// TwinCAT 3 PLC project rplc
// Title: rplc
// Company: TcHaxx
// Author: densogiaichned
// ProjectVersion: 0.3.2.0
// Description: Invoke RPC methods.
// ProgramVersion: 3.1.4024.0
// libraries:
//   Tc2_Standard, * (Beckhoff Automation GmbH)
//   Tc2_System, * (Beckhoff Automation GmbH)
//   Tc3_Module, * (Beckhoff Automation GmbH)
//   TcUnit, * (www.tcunit.org)
// project tree:
//   DUTs/ ST_AdsStatus.TcDUT, ST_AnyType.TcDUT
//   GVLs/ GCL.TcGVL, Param_Args.TcGVL
//   ITFs/ I_ArgsBuffer.TcIO, I_RpcArguments.TcIO, I_RpcDynamicConfigAmsNetId.TcIO, I_RpcDynamicConfigAmsPort.TcIO, I_RpcDynamicConfigSymbolPath.TcIO, I_RpcDynamicConfig.TcIO, I_RpcDynamicConfigBuild.TcIO, I_RpcInvoke.TcIO, I_RpcReleaseHandle.TcIO
//   / PlcTaskUnitTest.TcTTO
//   POUs/ FB_RPC.TcPOU, FB_RPC_Dynamic.TcPOU, F_ToAnyType.TcPOU
//   POUs/internal/ FB_ArgumentsBuffer.TcPOU, FB_RpcConfig.TcPOU, FB_RpcBase.TcPOU, F_RpcSymbol.TcPOU (not stored)
//   TESTs/ FB_F_RpcSymbol_Tests.TcPOU, FB_F_ToAnyType_Tests.TcPOU, FB_RPC_Tests.TcPOU, FB_RPC_Dynamic_Tests.TcPOU, PRG_UnitTests.TcPOU
//   TESTs/Helper/ E_Mode.TcDUT, F_IncrementStep.TcPOU
// real-time tasks:
//   TASK PlcTask: cycle T#10ms, priority 20, ADS port 350
//   TASK PlcTaskUnitTest: cycle T#10ms, priority 1, ADS port 351
//   TASK PlcTaskRpcServer: cycle T#10ms, priority 21, ADS port 352
//   TASK PlcTaskRpcClient: cycle T#10ms, priority 22, ADS port 353

CONFIGURATION rplc
    RESOURCE PLC ON TwinCAT3
        TASK PlcTaskUnitTest(INTERVAL := T#10ms, PRIORITY := 1);
        PROGRAM PRG_UnitTests WITH PlcTaskUnitTest : PRG_UnitTests;
    END_RESOURCE
END_CONFIGURATION

// ---- DUTs/ST_AdsStatus.TcDUT
{attribute 'pack_mode' = '1'}
TYPE ST_AdsStatus :
STRUCT
	bBusy	: BOOL;
	bError	: BOOL;
	nError 	: UDINT;
END_STRUCT
END_TYPE

// ---- DUTs/ST_AnyType.TcDUT
{attribute 'pack_mode' = '1'}
TYPE ST_AnyType :
STRUCT
	pValue : PVOID;
	nSize  : DINT;
	TypeClass : __SYSTEM.TYPE_CLASS;
END_STRUCT
END_TYPE

// ---- TESTs/Helper/E_Mode.TcDUT
{attribute 'qualified_only'}
{attribute 'strict'}
TYPE E_Mode :
(
	BUSY := 0,
	INC := 1,
	END := 99
);
END_TYPE

// ---- GVLs/GCL.TcGVL
{attribute 'qualified_only'}
{attribute 'no-analysis'}
{attribute 'global_init_slot' := '49991'}
VAR_GLOBAL CONSTANT
	cLocalAmsNetId		: STRING := '127.0.0.1.1.1';
	cAdsTimeOut			: TIME := Tc2_System.DEFAULT_ADS_TIMEOUT;
	cRpcSymbolSeparator : STRING := '#';
END_VAR

// ---- GVLs/Param_Args.TcGVL
{attribute 'qualified_only'}
{attribute 'no-analysis'}
VAR_GLOBAL CONSTANT
	cMaxArgsBuffer		: UDINT(64..1048576) 	:= 65536;	// max sizeof aArgs buffer array in bytes.
	cMaxArgs			: USINT(1..128) 		:= 32;		// max length method arguments
END_VAR

// ---- ITFs/I_ArgsBuffer.TcIO
INTERFACE I_ArgsBuffer

PROPERTY nArgsLength : UDINT
GET
END_GET
END_PROPERTY

PROPERTY nRetValLength : UDINT
GET
END_GET
END_PROPERTY

PROPERTY pArgsBuffer : POINTER TO BYTE
GET
END_GET
END_PROPERTY

PROPERTY pRetValBuffer : POINTER TO BYTE
GET
END_GET
END_PROPERTY

END_INTERFACE

// ---- ITFs/I_RpcArguments.TcIO
INTERFACE I_RpcArguments

METHOD NoReturnValue : I_RpcInvoke
VAR_INPUT
END_VAR
END_METHOD

METHOD ReturnValue : I_RpcInvoke
VAR_INPUT
	anyRetVal	: ANY;
END_VAR
END_METHOD

METHOD VarInOut : I_RpcArguments
VAR_INPUT
	anyArg	: ANY;
END_VAR
END_METHOD

METHOD VarInput : I_RpcArguments
VAR_INPUT
	anyArg	: ANY;
END_VAR
END_METHOD

METHOD VarOutput : I_RpcArguments
VAR_INPUT
	anyArg	: ANY;
END_VAR
END_METHOD

END_INTERFACE

// ---- ITFs/I_RpcDynamicConfigAmsNetId.TcIO
INTERFACE I_RpcDynamicConfigAmsNetId

METHOD WithAmsNetId : I_RpcDynamicConfigAmsPort
VAR_INPUT
	sAmsNetId	: T_AmsNetID;
END_VAR
END_METHOD

END_INTERFACE

// ---- ITFs/I_RpcDynamicConfigAmsPort.TcIO
INTERFACE I_RpcDynamicConfigAmsPort

METHOD WithAmsPort : I_RpcDynamicConfigSymbolPath
VAR_INPUT
	nAmsPort	: T_AmsPort;
END_VAR
END_METHOD

END_INTERFACE

// ---- ITFs/I_RpcDynamicConfigSymbolPath.TcIO
INTERFACE I_RpcDynamicConfigSymbolPath

METHOD WithSymbolPath : I_RpcDynamicConfigBuild
VAR_INPUT
	sInstancePath	: STRING;
	sSymbol			: STRING;
END_VAR
END_METHOD

END_INTERFACE

// ---- ITFs/I_RpcDynamicConfig.TcIO
INTERFACE I_RpcDynamicConfig

METHOD Configure : I_RpcDynamicConfigAmsNetId
VAR_INPUT
END_VAR
END_METHOD

END_INTERFACE

// ---- ITFs/I_RpcDynamicConfigBuild.TcIO
INTERFACE I_RpcDynamicConfigBuild

METHOD Build : HRESULT
VAR_INPUT
END_VAR
END_METHOD

END_INTERFACE

// ---- ITFs/I_RpcInvoke.TcIO
INTERFACE I_RpcInvoke

METHOD Invoke : ST_AdsStatus
VAR_INPUT
END_VAR
END_METHOD

END_INTERFACE

// ---- ITFs/I_RpcReleaseHandle.TcIO
INTERFACE I_RpcReleaseHandle

METHOD ReleaseHandle : ST_AdsStatus
VAR_INPUT
END_VAR
END_METHOD

END_INTERFACE

// ---- TESTs/PRG_UnitTests.TcPOU
{attribute 'analysis' := '-33'}
PROGRAM INTERNAL PRG_UnitTests

VAR
{IF defined (UNIT_TEST)}	
	fbF_RpcSymbolTests			: FB_F_RpcSymbol_Tests;
	fbRpcTests					: FB_RPC_Tests;
	fbRpcDynamicTests			: FB_RPC_Dynamic_Tests;
	fbF_ToAnyTypeTests			: FB_F_ToAnyType_Tests;
{END_IF}
END_VAR

{IF defined (UNIT_TEST)}
TcUnit.RUN();
{END_IF}

END_PROGRAM

// ---- TESTs/FB_F_RpcSymbol_Tests.TcPOU
{attribute 'reflection'}
FUNCTION_BLOCK INTERNAL FINAL FB_F_RpcSymbol_Tests EXTENDS TcUnit.FB_TestSuite
VAR_INPUT
END_VAR
VAR_OUTPUT
END_VAR
VAR
	{attribute 'instance-path'} 
    {attribute 'noinit'} 
	sTestName			: T_MaxString;
	sActual				: T_MaxString;
	sMaxString			: T_MaxString := 'iwgNivAMcHfLkBpkvqNXNWYnMrQNVzUhZFVRYSjRcjnJtRacqFJhzGPkUNrHkvVpMnnxcBtbBwcrvBgfHgaLBQffiYTVjMkCQgidjvwmnvQEQCzVzZUguBPbnEQCfVDbiCMwiEdfqETncfBwbYbhTrSuRhWzNxVpQzBiWeHAGjdWTLmVfyFKEWMhmMgWqFvtAhBarrEkqQCMJvWxGcDZUfMZwdEebgjfuXXMJwGbgzpjyqzigwxkZiHXPvZCmcn';
END_VAR


TEST(sTestName);

TEST('Should build RPC symbol successfully');

sActual := F_RpcSymbol('', '');
AssertEquals_STRING(Expected:= GCL.cRpcSymbolSeparator,
					Actual:= sActual,
					Message:= 'Expected # only');

sActual := F_RpcSymbol('abc', '');
AssertEquals_STRING(Expected:= 'abc#',
					Actual:= sActual,
					Message:= 'Expected abc# only');

sActual := F_RpcSymbol('', 'abc');
AssertEquals_STRING(Expected:= '#abc',
					Actual:= sActual,
					Message:= 'Expected #abc only');

sActual := F_RpcSymbol('InstancePath', 'SymbolName');
AssertEquals_STRING(Expected:= 'InstancePath#SymbolName',
					Actual:= sActual,
					Message:= 'Expected InstancePath#SymbolName');
TEST_FINISHED();

TEST('Should return sInstancePath if > T_MaxString');

sActual := F_RpcSymbol(sMaxString, 'abc');
AssertEquals_STRING(Expected:= sMaxString,
					Actual:= sActual,
					Message:= 'Expected sInstancePath');
TEST_FINISHED();

TEST('Should truncate if > T_MaxString');


sActual := F_RpcSymbol('abc', sMaxString);
AssertEquals_STRING(Expected:= CONCAT('abc#', LEFT(sMaxString, 251)),
					Actual:= sActual,
					Message:= 'Expected abc#iwgNivAMcHfLk...ZiHXPvZ');
TEST_FINISHED();

TEST_FINISHED_NAMED(sTestName);

END_FUNCTION_BLOCK

// ---- TESTs/FB_RPC_Tests.TcPOU
{attribute 'reflection'}
FUNCTION_BLOCK INTERNAL FINAL FB_RPC_Tests EXTENDS TcUnit.FB_TestSuite
VAR
	{attribute 'instance-path'} 
    {attribute 'noinit'} 
	sTestName			: T_MaxString;
	sActiveStep			: T_MaxString;
	nSequence			: INT;
	nSeqOld				: INT;
	nRpcMethodInvoked 	: UDINT;
	aSUTs				: ARRAY[0..255] OF I_RpcReleaseHandle;
END_VAR
VAR_TEMP
	eMode	: E_Mode;
END_VAR

CASE nSequence OF
	0:
		TEST(sTestName);
		F_IncrementStep(nStepToInc:= nSequence, sActiveStep:= sActiveStep, eMode:= E_Mode.INC);
	1:
		sActiveStep := 'ShouldInvokeMethod_NoArguments_NoReturnValue_Successfully';
		TEST(sActiveStep);
		eMode := ShouldInvokeMethod_NoArguments_NoReturnValue_Successfully();
		F_IncrementStep(nStepToInc:= nSequence, sActiveStep, eMode);
	2:
		sActiveStep := 'ShouldInvokeMethod_NoArguments_ReturnValueBoolean_Successfully';
		TEST(sActiveStep);
		eMode := ShouldInvokeMethod_NoArguments_ReturnValueBoolean_Successfully();
		F_IncrementStep(nStepToInc:= nSequence, sActiveStep, eMode);
	3:	
		sActiveStep := 'ShouldInvokeMethod_OneArgument_NoReturnValue_Successfully';
		TEST(sActiveStep);
		eMode := ShouldInvokeMethod_OneArgument_NoReturnValue_Successfully();
		F_IncrementStep(nStepToInc:= nSequence, sActiveStep, eMode);	
	4:	
		sActiveStep := 'ShouldInvokeMethod_OneArgument_NoReturnValue_Successfully';
		TEST(sActiveStep);
		eMode := ShouldInvokeMethod_OneArgument_NoReturnValue_Successfully();
		F_IncrementStep(nStepToInc:= nSequence, sActiveStep, eMode);	
	5:	
		sActiveStep := 'ShouldInvokeMethod_TwoArguments_ReturnValue_Successfully';
		TEST(sActiveStep);
		eMode := ShouldInvokeMethod_TwoArguments_ReturnValue_Successfully();
		F_IncrementStep(nStepToInc:= nSequence, sActiveStep, eMode);
	6:	
		sActiveStep := 'ShouldInvokeMethod_ThreeArguments_ReturnValue_Successfully';
		TEST(sActiveStep);
		eMode := ShouldInvokeMethod_ThreeArguments_ReturnValue_Successfully();
		F_IncrementStep(nStepToInc:= nSequence, sActiveStep, eMode);		
	7:	
		sActiveStep := 'ShouldInvokeMethod_VarInOutConstant_ReturnValue_Successfully';
		TEST(sActiveStep);
		eMode := ShouldInvokeMethod_VarInOutConstant_ReturnValue_Successfully();
		F_IncrementStep(nStepToInc:= nSequence, sActiveStep, eMode);	
	8:	
		sActiveStep := 'ShouldInvokeMethod_VarOutput_ReturnValue_Successfully';
		TEST(sActiveStep);
		eMode := ShouldInvokeMethod_VarOutput_ReturnValue_Successfully();
		F_IncrementStep(nStepToInc:= nSequence, sActiveStep, eMode);	
	9:	
		sActiveStep := 'ShouldInvokeMethod_TwoVarOutput_ReturnValue_Successfully';
		TEST(sActiveStep);
		eMode := ShouldInvokeMethod_TwoVarOutput_ReturnValue_Successfully();
		F_IncrementStep(nStepToInc:= nSequence, sActiveStep, eMode);	
	10:	
		sActiveStep := 'ShouldInvokeMethod_VarInput_VarInOut_VarOutput_ReturnValue_Successfully';
		TEST(sActiveStep);
		eMode := ShouldInvokeMethod_VarInput_VarInOut_VarOutput_ReturnValue_Successfully();
		F_IncrementStep(nStepToInc:= nSequence, sActiveStep, eMode);		
	11: 
		sActiveStep := 'ShouldReturnError0x705';
		TEST(sActiveStep);
		eMode := ShouldReturnError0x705();
		F_IncrementStep(nStepToInc:= nSequence, sActiveStep, eMode);	
	12: 
		sActiveStep := 'ShouldReturnError0x710';
		TEST(sActiveStep);
		eMode := ShouldReturnError0x710();
		F_IncrementStep(nStepToInc:= nSequence, sActiveStep, eMode);	
	13: 
		sActiveStep := 'ShouldReleaseAllSymbolHandleSuccessfully';
		TEST(sActiveStep);
		eMode := ShouldReleaseAllSymbolHandleSuccessfully();
		F_IncrementStep(nStepToInc:= nSequence, sActiveStep, eMode);	
	ELSE
		TEST_FINISHED_NAMED(sTestName);
END_CASE

IF nSequence <> nSeqOld THEN
	nRpcMethodInvoked := 0;
	nSeqOld := nSequence;
END_IF;

{attribute 'TcRpcEnable'}
METHOD NoParameter_NoReturnValue

nRpcMethodInvoked := nRpcMethodInvoked + 1;
END_METHOD

{attribute 'TcRpcEnable'}
METHOD NoParameter_ReturnValue : BOOL
VAR_INPUT
END_VAR
nRpcMethodInvoked := nRpcMethodInvoked + 1;
NoParameter_ReturnValue := nRpcMethodInvoked > 0;
END_METHOD

{attribute 'TcRpcEnable'}
METHOD OneParameter_NoReturnValue
VAR_INPUT
	nArg1 	: UDINT;
END_VAR
nRpcMethodInvoked := nArg1;
END_METHOD

METHOD Register
VAR_INPUT
	ipRpcReleaseHandle	: I_RpcReleaseHandle;
END_VAR

VAR
	i :UINT;
END_VAR


FOR i:=0 TO 255 DO	
	IF aSUTs[i] = ipRpcReleaseHandle THEN
		EXIT;
	END_IF
	IF aSUTs[i] <> NULL THEN
		CONTINUE;
	END_IF
	
	aSUTs[i] := ipRpcReleaseHandle;
	EXIT;
END_FOR
END_METHOD

METHOD ShouldInvokeMethod_NoArguments_NoReturnValue_Successfully : E_Mode

VAR_INST
	fbSUT		: FB_RPC(GCL.cLocalAmsNetId, _AppInfo.AdsPort, 'PRG_UnitTests.fbRpcTests', 'NoParameter_NoReturnValue');
END_VAR

VAR
	stRetVal	: ST_AdsStatus;
	eMode		: E_Mode := E_MODE.BUSY;
END_VAR
// Arrange
Register(fbSUT);

// Act
stRetVal := fbSUT.Invoke();

IF NOT stRetVal.bBusy THEN
	eMode := E_Mode.INC;
	
	// Assert
	AssertFalse(Condition:= stRetVal.bError, Message:= 'Expected method NoParameter_NoReturnValue to return no error.');
	AssertEquals_UDINT(Expected:= E_AdsErr.NOERR, Actual:= stRetVal.nError, Message:= 'Expected method NoParameter_NoReturnValue to return no error.');
	AssertEquals_UDINT(Expected:= 1, Actual:= nRpcMethodInvoked, Message:= 'Expected method NoParameter_NoReturnValue to be invoked once.');
END_IF

ShouldInvokeMethod_NoArguments_NoReturnValue_Successfully := eMode;
END_METHOD

METHOD ShouldInvokeMethod_NoArguments_ReturnValueBoolean_Successfully : E_Mode

VAR_INST
	fbSUT		: FB_RPC(GCL.cLocalAmsNetId, _AppInfo.AdsPort, 'PRG_UnitTests.fbRpcTests', 'NoParameter_ReturnValue');
END_VAR

VAR
	stRetVal	: ST_AdsStatus;
	eMode		: E_Mode := E_MODE.BUSY;
	bActual		: BOOL;
END_VAR
// Arrange
Register(fbSUT);

// Act
stRetVal := fbSUT.ReturnValue(bActual).Invoke();

IF NOT stRetVal.bBusy THEN
	eMode := E_Mode.INC;
	// Assert
	AssertFalse(Condition:= stRetVal.bError, Message:= 'Expected method NoParameter_ReturnValue to return no error.');
	AssertEquals_UDINT(Expected:= E_AdsErr.NOERR, Actual:= stRetVal.nError, Message:= 'Expected method NoParameter_ReturnValue to return no error.');
	AssertEquals_UDINT(Expected:= 1, Actual:= nRpcMethodInvoked, Message:= 'Expected method NoParameter_ReturnValue to be invoked once.');
	AssertTrue(Condition:= bActual, Message:= 'Expected method NoParameter_ReturnValue to return TRUE.');
END_IF

ShouldInvokeMethod_NoArguments_ReturnValueBoolean_Successfully := eMode;
END_METHOD

METHOD ShouldInvokeMethod_OneArgument_NoReturnValue_Successfully : E_Mode

VAR_INST
	fbSUT		: FB_RPC(GCL.cLocalAmsNetId, _AppInfo.AdsPort, 'PRG_UnitTests.fbRpcTests', 'OneParameter_NoReturnValue');
END_VAR

VAR
	stRetVal	: ST_AdsStatus;
	eMode		: E_Mode := E_MODE.BUSY;
	nArg		: UDINT;
END_VAR
// Arrange
Register(fbSUT);
nArg := 123;

// Act
stRetVal := fbSUT.VarInput(nArg).NoReturnValue().Invoke();

IF NOT stRetVal.bBusy THEN
	eMode := E_Mode.INC;
	
	// Assert
	AssertFalse(Condition:= stRetVal.bError, Message:= 'Expected method OneParameter_NoReturnValue to return no error.');
	AssertEquals_UDINT(Expected:= E_AdsErr.NOERR, Actual:= stRetVal.nError, Message:= 'Expected method OneParameter_NoReturnValue to return no error.');
	AssertEquals_UDINT(Expected:= nArg, Actual:= nRpcMethodInvoked, Message:= 'Expected method OneParameter_NoReturnValue to be invoked with value 123.');
END_IF

ShouldInvokeMethod_OneArgument_NoReturnValue_Successfully := eMode;
END_METHOD

METHOD ShouldInvokeMethod_ThreeArguments_ReturnValue_Successfully : E_Mode

VAR_INST
	fbSUT		: FB_RPC(GCL.cLocalAmsNetId, _AppInfo.AdsPort, 'PRG_UnitTests.fbRpcTests', 'ThreeParameters_ReturnValue');
END_VAR

VAR
	stRetVal	: ST_AdsStatus;
	eMode		: E_Mode := E_MODE.BUSY;
	nArg1		: UDINT;
	stArg2		: ST_AdsStatus;	// IN_OUT!
	sArg3		: STRING;
	sActualRetVal : STRING;
END_VAR
// Arrange
Register(fbSUT);
nArg1 := 456;
stArg2.bBusy := FALSE;
stArg2.bError := TRUE;
stArg2.nError := 321;
sArg3 := 'third Argument';

// Act
stRetVal := fbSUT.VarInput(nArg1).VarInOut(stArg2).VarInput(sArg3).ReturnValue(sActualRetVal).Invoke();

IF NOT stRetVal.bBusy THEN
	eMode := E_Mode.INC;
	
	// Assert
	AssertFalse(Condition:= stRetVal.bError, Message:= 'Expected method TwoParameters_ReturnValue to return no error.');
	AssertEquals_UDINT(Expected:= E_AdsErr.NOERR, Actual:= stRetVal.nError, Message:= 'Expected method ThreeParameters_ReturnValue to return no error.');
	AssertEquals_UDINT(Expected:= nArg1, Actual:= nRpcMethodInvoked, Message:= 'Expected method ThreeParameters_ReturnValue to be invoked with value 456.');
	AssertTrue(Condition:= stArg2.bBusy, Message:= 'Expected method ThreeParameters_ReturnValue to invert bBusy of VAR_IN_OUT');
	AssertFalse(Condition:= stArg2.bError, Message:= 'Expected method ThreeParameters_ReturnValue to invert bError of VAR_IN_OUT');
	AssertEquals_UDINT(Expected:= 321 * 2, Actual:= stArg2.nError, Message:= 'Expected method ThreeParameters_ReturnValue to double value nError of VAR_IN_OUT');
	AssertEquals_STRING(Expected:= sArg3, Actual:= sActualRetVal, Message:= 'Expected method ThreeParameters_ReturnValue to return value .');
END_IF

ShouldInvokeMethod_ThreeArguments_ReturnValue_Successfully := eMode;
END_METHOD

METHOD ShouldInvokeMethod_TwoArguments_ReturnValue_Successfully : E_Mode

VAR_INST
	fbSUT		: FB_RPC(GCL.cLocalAmsNetId, _AppInfo.AdsPort, 'PRG_UnitTests.fbRpcTests', 'TwoParameters_ReturnValue');
END_VAR

VAR
	stRetVal	: ST_AdsStatus;
	eMode		: E_Mode := E_MODE.BUSY;
	nArg1		: UDINT;
	sArg2		: STRING;
	sActualRetVal : STRING;
END_VAR
// Arrange
Register(fbSUT);
nArg1 := 456;
sArg2 := 'second Argument';

// Act
stRetVal := fbSUT.VarInput(nArg1).VarInput(sArg2).ReturnValue(sActualRetVal).Invoke();

IF NOT stRetVal.bBusy THEN
	eMode := E_Mode.INC;
	
	// Assert
	AssertFalse(Condition:= stRetVal.bError, Message:= 'Expected method TwoParameters_ReturnValue to return no error.');
	AssertEquals_UDINT(Expected:= E_AdsErr.NOERR, Actual:= stRetVal.nError, Message:= 'Expected method TwoParameters_ReturnValue to return no error.');
	AssertEquals_UDINT(Expected:= nArg1, Actual:= nRpcMethodInvoked, Message:= 'Expected method TwoParameters_ReturnValue to be invoked with value 456.');
	AssertEquals_STRING(Expected:= sArg2, Actual:= sActualRetVal, Message:= 'Expected method TwoParameters_ReturnValue to return value .');
END_IF

ShouldInvokeMethod_TwoArguments_ReturnValue_Successfully := eMode;
END_METHOD

METHOD ShouldInvokeMethod_TwoVarOutput_ReturnValue_Successfully : E_Mode

VAR_INST
	fbSUT		: FB_RPC(GCL.cLocalAmsNetId, _AppInfo.AdsPort, 'PRG_UnitTests.fbRpcTests', 'TwoVarOutput_ReturnValue');
END_VAR

VAR
	stRetVal	: ST_AdsStatus;
	eMode		: E_Mode := E_MODE.BUSY;
	stArg		: ST_AdsStatus;
	nA			: UDINT;
	nActualRetVal : UDINT;
END_VAR
// Arrange
Register(fbSUT);

// Act
stRetVal := fbSUT.VarOutput(stArg).VarOutput(nA).ReturnValue(nActualRetVal).Invoke();

IF NOT stRetVal.bBusy THEN
	eMode := E_Mode.INC;
	
	// Assert
	AssertFalse(Condition:= stRetVal.bError, Message:= 'Expected method VarOutput_ReturnValue to return no error.');
	AssertEquals_UDINT(Expected:= E_AdsErr.NOERR, Actual:= stRetVal.nError, Message:= 'Expected method VarOutput_ReturnValue to return no error.');
	AssertFalse(Condition:= stArg.bBusy, Message:= 'Expected method VarOutput_ReturnValue to return stArg.bBusy = FALSE');
	AssertTrue(Condition:= stArg.bError, Message:= 'Expected method VarOutput_ReturnValue to return stArg.bError = TRUE');
	AssertEquals_UDINT(Expected:= 123, Actual:= stARg.nError, Message:= 'Expected method VarOutput_ReturnValue to return stArg.nError = 123');
	AssertEquals_UDINT(Expected:= 789, Actual:= nA, Message:= 'Expected method VarOutput_ReturnValue to return nA = 789');
	AssertEquals_UDINT(Expected:= 456, Actual:= nActualRetVal, Message:= 'Expected method VarOutput_ReturnValue to return 456.');
END_IF

ShouldInvokeMethod_TwoVarOutput_ReturnValue_Successfully := eMode;
END_METHOD

METHOD ShouldInvokeMethod_VarInOutConstant_ReturnValue_Successfully : E_Mode

VAR_INST
	fbSUT		: FB_RPC(GCL.cLocalAmsNetId, _AppInfo.AdsPort, 'PRG_UnitTests.fbRpcTests', 'VarInOutConstant_ReturnValue');
END_VAR

VAR
	stRetVal	: ST_AdsStatus;
	eMode		: E_Mode := E_MODE.BUSY;
	stArg		: ST_LibVersion;
	nActualRetVal : UDINT;
END_VAR
// Arrange
Register(fbSUT);
stArg.nFlags := 987;

// Act
stRetVal := fbSUT.VarInOut(stArg).ReturnValue(nActualRetVal).Invoke();

IF NOT stRetVal.bBusy THEN
	eMode := E_Mode.INC;
	
	// Assert
	AssertFalse(Condition:= stRetVal.bError, Message:= 'Expected method VarInOutConstant_ReturnValue to return no error.');
	AssertEquals_UDINT(Expected:= E_AdsErr.NOERR, Actual:= stRetVal.nError, Message:= 'Expected method VarInOutConstant_ReturnValue to return no error.');
	AssertEquals_DWORD(Expected:= 987, Actual:= stArg.nFlags, Message:= 'Expected method VarInOutConstant_ReturnValue to be invoked with value 987.');
	AssertEquals_UDINT(Expected:= 987, Actual:= nActualRetVal, Message:= 'Expected method VarInOutConstant_ReturnValue to be invoked with value 987.');
END_IF

ShouldInvokeMethod_VarInOutConstant_ReturnValue_Successfully := eMode;
END_METHOD

METHOD ShouldInvokeMethod_VarInput_VarInOut_VarOutput_ReturnValue_Successfully : E_Mode

VAR_INST
	fbSUT		: FB_RPC(GCL.cLocalAmsNetId, _AppInfo.AdsPort, 'PRG_UnitTests.fbRpcTests', 'VarInput_VarInOut_VarOutput_ReturnValue');
END_VAR

VAR
	stRetVal	: ST_AdsStatus;
	eMode		: E_Mode := E_MODE.BUSY;
		
	sStrIn		: STRING;
	nIn			: INT;
	nInOut 		: INT;
	stArgOut	: ST_AdsStatus;
	sStrOut		: STRING;	
	sRetVal		: STRING;
END_VAR
// Arrange
Register(fbSUT);

sStrIn	:= 'Input String';
nIn		:= -666;
nInOut	:= 777;

// Act
stRetVal := fbSUT.VarInput(sStrIn).VarInput(nIn).VarInOut(nInOut).VarOutput(stArgOut).VarOutput(sStrOut).ReturnValue(sRetVal).Invoke();

IF NOT stRetVal.bBusy THEN
	eMode := E_Mode.INC;
	
	// Assert
	AssertFalse(Condition:= stRetVal.bError, Message:= 'Expected method VarInput_VarInOut_VarOutput_ReturnValue to return no error.');
	AssertEquals_UDINT(Expected:= E_AdsErr.NOERR, Actual:= stRetVal.nError, Message:= 'Expected method VarInput_VarInOut_VarOutput_ReturnValue to return no error.');
	AssertTrue(Condition:= stArgOut.bBusy, Message:= 'Expected method VarInput_VarInOut_VarOutput_ReturnValue to return stArgOut.bBusy = TRUE');
	AssertFalse(Condition:= stArgOut.bError, Message:= 'Expected method VarInput_VarInOut_VarOutput_ReturnValue to return stArgOut.bError = FALSE');
	AssertEquals_UDINT(Expected:= 222, Actual:= stArgOut.nError, Message:= 'Expected method VarInput_VarInOut_VarOutput_ReturnValue to return stArgOut.nError = 222');
	AssertEquals_STRING(Expected:= 'sStrOut: Input String', Actual:= sStrOut,
						Message:= 'Expected method VarInput_VarInOut_VarOutput_ReturnValue to return "sStrOut: Input String"');
	AssertEquals_STRING(Expected:= 'ReturnValue: Input String', Actual:= sRetVal,
						Message:= 'Expected method VarInput_VarInOut_VarOutput_ReturnValue to return "ReturnValue: Input String"');
END_IF

ShouldInvokeMethod_VarInput_VarInOut_VarOutput_ReturnValue_Successfully := eMode;
END_METHOD

METHOD ShouldInvokeMethod_VarOutput_ReturnValue_Successfully : E_Mode

VAR_INST
	fbSUT		: FB_RPC(GCL.cLocalAmsNetId, _AppInfo.AdsPort, 'PRG_UnitTests.fbRpcTests', 'VarOutput_ReturnValue');
END_VAR

VAR
	stRetVal	: ST_AdsStatus;
	eMode		: E_Mode := E_MODE.BUSY;
	stArg		: ST_AdsStatus;
	nActualRetVal : UDINT;
END_VAR
// Arrange
Register(fbSUT);


// Act
stRetVal := fbSUT.VarOutput(stArg).ReturnValue(nActualRetVal).Invoke();

IF NOT stRetVal.bBusy THEN
	eMode := E_Mode.INC;
	
	// Assert
	AssertFalse(Condition:= stRetVal.bError, Message:= 'Expected method VarOutput_ReturnValue to return no error.');
	AssertEquals_UDINT(Expected:= E_AdsErr.NOERR, Actual:= stRetVal.nError, Message:= 'Expected method VarOutput_ReturnValue to return no error.');
	AssertTrue(Condition:= stArg.bBusy, Message:= 'Expected method VarOutput_ReturnValue to return bBusy = TRUE.');
	AssertFalse(Condition:= stArg.bError, Message:= 'Expected method VarOutput_ReturnValue to return bError = FALSE');
	AssertEquals_UDINT(Expected:= 456, Actual:= stARg.nError, Message:= 'Expected method VarOutput_ReturnValue to return VAR_OUTPUT 456.');
	AssertEquals_UDINT(Expected:= 123, Actual:= nActualRetVal, Message:= 'Expected method VarOutput_ReturnValue to return 123.');
END_IF

ShouldInvokeMethod_VarOutput_ReturnValue_Successfully := eMode;
END_METHOD

METHOD ShouldReleaseAllSymbolHandleSuccessfully : E_Mode

VAR
	stRetVal	: ST_AdsStatus;
	ipSUT		: I_RpcReleaseHandle;
END_VAR

VAR_INST
	nIndex 		: UINT := 0;
END_VAR


ipSUT := aSUTs[nIndex];
IF ipSUT = NULL THEN
	ShouldReleaseAllSymbolHandleSuccessfully := E_Mode.INC;
	RETURN;
END_IF

// Act
stRetVal := ipSUT.ReleaseHandle();

IF NOT stRetVal.bBusy THEN
	nIndex := nIndex + 1;	
	// Assert
	AssertFalse(Condition:= stRetVal.bError, Message:= 'Expected ReleaseHandle to return no error.');
	AssertEquals_UDINT(Expected:= E_AdsErr.NOERR, Actual:= stRetVal.nError, Message:= 'Expected ReleaseHandle to return no error.');
END_IF

ShouldReleaseAllSymbolHandleSuccessfully := E_Mode.BUSY;
END_METHOD

METHOD ShouldReturnError0x705 : E_Mode

VAR_INST
	fbSUT		: FB_RPC(GCL.cLocalAmsNetId, _AppInfo.AdsPort, 'PRG_UnitTests.fbRpcTests', 'NoParameter_NoReturnValue');
END_VAR

VAR
	stRetVal	: ST_AdsStatus;
	eMode		: E_Mode := E_MODE.BUSY;
	nDummy		: INT;
END_VAR
// Act
stRetVal := fbSUT.VarInput(nDummy).NoReturnValue().Invoke();

IF NOT stRetVal.bBusy THEN
	eMode := E_Mode.INC;
	
	// Assert
	AssertTrue(Condition:= stRetVal.bError, Message:= 'Expected method NoParameter_NoReturnValue to return error.');
	AssertEquals_UDINT(Expected:= E_AdsErr.DEVICE_INVALIDSIZE, Actual:= stRetVal.nError, Message:= 'Expected method NoParameter_NoReturnValue to return error ADSERR_DEVICE_INVALIDSIZE.');
	AssertEquals_UDINT(Expected:= 0, Actual:= nRpcMethodInvoked, Message:= 'Expected method NoParameter_NoReturnValue to not be invoked.');
END_IF

ShouldReturnError0x705 := eMode;
END_METHOD

METHOD ShouldReturnError0x710 : E_Mode

VAR_INST
	fbSUT		: FB_RPC(GCL.cLocalAmsNetId, _AppInfo.AdsPort, 'PRG_UnitTests.fbRpcTests', 'NotExistingSymbol');
END_VAR

VAR
	stRetVal	: ST_AdsStatus;
	eMode		: E_Mode := E_MODE.BUSY;
	nDummy		: INT;
END_VAR
// Act
stRetVal := fbSUT.VarInput(nDummy).NoReturnValue().Invoke();

IF NOT stRetVal.bBusy THEN
	eMode := E_Mode.INC;
	
	// Assert
	AssertTrue(Condition:= stRetVal.bError, Message:= 'Expected return error.');
	AssertEquals_UDINT(Expected:= E_AdsErr.DEVICE_SYMBOLNOTFOUND, Actual:= stRetVal.nError, Message:= 'Expected error ADSERR_DEVICE_SYMBOLNOTFOUND.');
END_IF

ShouldReturnError0x710 := eMode;
END_METHOD

{attribute 'TcRpcEnable'}
METHOD ThreeParameters_ReturnValue : STRING
VAR_INPUT
	nArg1 	: UDINT;
END_VAR
VAR_IN_OUT
	stArg2  : ST_AdsStatus;
END_VAR
VAR_INPUT
	sArg3	: STRING;
END_VAR
nRpcMethodInvoked := nArg1;
stArg2.bBusy := NOT stArg2.bBusy;
stArg2.bError := NOT stARg2.bError;
stARg2.nError := stARg2.nError * 2;
ThreeParameters_ReturnValue := sArg3;
END_METHOD

{attribute 'TcRpcEnable'}
METHOD TwoParameters_ReturnValue : STRING
VAR_INPUT
	nArg1 	: UDINT;
	sArg2	: STRING;
END_VAR
nRpcMethodInvoked := nArg1;
TwoParameters_ReturnValue := sArg2;
END_METHOD

{attribute 'TcRpcEnable'}
METHOD TwoVarOutput_ReturnValue : UDINT
VAR_OUTPUT
	stArg	: ST_AdsStatus;
	nA		: UDINT;
END_VAR

stArg.bBusy := FALSE;
stArg.bError := TRUE;
stArg.nError := 123;
nA := 789;
TwoVarOutput_ReturnValue := 456;
END_METHOD

{attribute 'TcRpcEnable'}
METHOD VarInOutConstant_ReturnValue : DWORD
VAR_IN_OUT CONSTANT
	stArg  : ST_LibVersion;
END_VAR
VarInOutConstant_ReturnValue := stArg.nFlags;
END_METHOD

{attribute 'TcRpcEnable'}
METHOD VarInput_VarInOut_VarOutput_ReturnValue : STRING
VAR_INPUT
	sStrIn	: STRING;
	nIn		: INT;
END_VAR
VAR_IN_OUT
	nInOut	: INT;	
END_VAR
VAR_OUTPUT
	stArgOut	: ST_AdsStatus;
	sStrOut 	: STRING;
END_VAR



nInOut := nInOut + nIn;

stArgOut.bBusy := TRUE;
stArgOut.bError := FALSE;
stArgOut.nError := 222;

sStrOut := CONCAT('sStrOut: ',sStrIn);

VarInput_VarInOut_VarOutput_ReturnValue := CONCAT('ReturnValue: ',sStrIn);
END_METHOD

{attribute 'TcRpcEnable'}
METHOD VarOutput_ReturnValue : UDINT
VAR_OUTPUT
	stArg  : ST_AdsStatus;
END_VAR

stArg.bBusy := TRUE;
stArg.bError := FALSE;
stArg.nError := 456;
VarOutput_ReturnValue := 123;
END_METHOD

END_FUNCTION_BLOCK

// ---- TESTs/Helper/F_IncrementStep.TcPOU
FUNCTION INTERNAL F_IncrementStep
VAR_IN_OUT
	nStepToInc : INT; 
END_VAR
VAR_IN_OUT CONSTANT
	sActiveStep : T_MaxString; 
END_VAR
VAR_INPUT
	eMode : E_Mode;
END_VAR
VAR CONSTANT
	cStepFinished : INT := -999;
END_VAR

CASE eMode OF
	E_Mode.BUSY:
		RETURN;
	E_Mode.INC:
		nStepToInc := nStepToInc + 1;
		IF sActiveStep <> '' THEN
			TEST_FINISHED_NAMED(sActiveStep);
		END_IF
	E_Mode.END:
		nStepToInc := cStepFinished;
		IF sActiveStep <> '' THEN
			TEST_FINISHED_NAMED(sActiveStep);
		END_IF
END_CASE

END_FUNCTION

// ---- POUs/FB_RPC.TcPOU
{attribute 'no_explicit_call' := 'do not call this POU directly'}
{attribute 'conditionalshow_all_locals'}
// Function Block to invoke RPC calls.
FUNCTION_BLOCK FINAL FB_RPC EXTENDS FB_RpcBase

VAR
END_VAR

{attribute 'no-analysis'}
METHOD INTERNAL ConfigDoneCallback : HRESULT
VAR_INPUT CONSTANT
	sAmsNetId		: REFERENCE TO T_AmsNetId;
	nAmsPort		: T_AmsPort;
	sInstancePath	: REFERENCE TO STRING;
	sSymbol			: REFERENCE TO STRING;
END_VAR
ConfigDoneCallback := S_FALSE;
END_METHOD

METHOD FB_exit : BOOL
VAR_INPUT
	bInCopyCode : BOOL; // if TRUE, the exit method is called for exiting an instance that is copied afterwards (online change).
END_VAR
IF SUPER^.nSymbolHandle > cNoSymbolNameHandle THEN
	SUPER^.ReleaseHandle();
END_IF
END_METHOD

METHOD FB_init : BOOL
VAR_INPUT
    bInitRetains 	: BOOL; // if TRUE, the retain variables are initialized (warm start / cold start)
    bInCopyCode  	: BOOL; // if TRUE, the instance afterwards gets moved into the copy code (online change)
	sAmsNetId		: T_AmsNetID;
	nAmsPort		: T_AmsPort;
	sInstancePath	: STRING;	// e.g. MAIN.fbYourFB
	sSymbol			: STRING;	// e.g. YourSymbolName
END_VAR
SUPER^.Reset();

IF bInCopyCode THEN
	SUPER^.ReleaseHandle();
END_IF


IF sAmsNetId = '' THEN
	SUPER^.sAmsNetId := GCL.cLocalAmsNetId;
ELSE
	SUPER^.sAmsNetId := sAmsNetId;
END_IF

SUPER^.nAmsPort := nAmsPort;

SUPER^.sRpcSymbol := F_RpcSymbol(sInstancePath, sSymbol);
END_METHOD

END_FUNCTION_BLOCK

// ---- POUs/internal/FB_RpcBase.TcPOU
{attribute 'no_explicit_call' := 'do not call this POU directly'}
{attribute 'conditionalshow_all_locals'}
FUNCTION_BLOCK INTERNAL ABSTRACT FB_RpcBase IMPLEMENTS I_RpcArguments, I_RpcInvoke, I_RpcReleaseHandle, __System.IQueryInterface
VAR
	sAmsNetIdField 			: T_AmsNetId 	:= GCL.cLocalAmsNetId;
	nAmsPortField			: T_AmsPort		:= 851;
	nSymbolHandle 			: UDINT;
	sRpcSymbolField			: T_MaxString	:= 'MAIN.NotInitialized#yet';
END_VAR
VAR
	fbRdWrReq 				: ADSRDWRT;
	fbAdsWrReqRelHandle 	: ADSWRITE; 
	nHandleToRelease		: UDINT := cNoSymbolNameHandle;	
	eStep					: ( HNDBYNAME, VALBYHND, RELEASEHND) := HNDBYNAME;
	eArgs					: ( NO_LOCK, LOCK ) := NO_LOCK;
	fbArguments				: FB_ArgumentsBuffer;
	tAdsTimeOutField		: TIME := GCL.cAdsTimeOut;
END_VAR

VAR CONSTANT
	cNoSymbolNameHandle : UDINT := 0;
END_VAR

METHOD INTERNAL ABSTRACT ConfigDoneCallback : HRESULT
VAR_INPUT CONSTANT
	sAmsNetId		: REFERENCE TO T_AmsNetId;
	nAmsPort		: T_AmsPort;
	sInstancePath	: REFERENCE TO STRING;
	sSymbol			: REFERENCE TO STRING;
END_VAR
END_METHOD

METHOD PRIVATE GetSymbolHandleByName : ST_AdsStatus
VAR_INPUT
	sNetId 		: REFERENCE TO T_AmsNetId;
	nPort		: T_AmsPort;
	sSymbol		: REFERENCE TO T_MaxString;
END_VAR
fbRdWrReq(
	NETID:= sNetId, 
	PORT:= nPort, 
	IDXGRP:= ADSIGRP_SYM_HNDBYNAME, 
	IDXOFFS:= 16#0, 
	WRITELEN:= TO_UDINT(LEN(sSymbol)), 
	READLEN:= SIZEOF(nSymbolHandle), 
	SRCADDR:= ADR(sSymbol), 
	DESTADDR:= ADR(nSymbolHandle), 
	WRTRD:= TRUE, 
	TMOUT:= tAdsTimeOutField, 
	BUSY=> GetSymbolHandleByName.bBusy, 
	ERR=> GetSymbolHandleByName.bError, 
	ERRID=> GetSymbolHandleByName.nError);
END_METHOD

METHOD Invoke : ST_AdsStatus

VAR
	stRetVal : ST_AdsStatus;
END_VAR
eArgs := LOCK;

CASE eStep OF
	HNDBYNAME:
		Invoke.bBusy := TRUE;
		stRetVal := GetSymbolHandleByName(sAmsNetIdField, nAmsPortField, sRpcSymbolField);
		IF NOT stRetVal.bBusy AND NOT stRetVal.bError THEN
			fbRdWrReq(WRTRD:= FALSE);
			eStep:= VALBYHND;
		ELSE
			Invoke := stRetVal;
			eStep := HNDBYNAME;
			RETURN;
		END_IF
		
	VALBYHND:
		Invoke := ReadValueByHandle(fbArguments.pArgsBuffer,
									fbArguments.nArgsLength, 
									fbArguments.pRetValBuffer, 
									fbArguments.nRetValLength);		
		IF NOT Invoke.bBusy THEN
			eArgs := NO_LOCK;
			IF NOT Invoke.bError THEN
				Invoke.nError := fbArguments.GetRetVal();
				Invoke.bError := Invoke.nError <> E_AdsErr.NOERR;
			END_IF;
			fbRdWrReq(WRTRD:= FALSE);
			ResetArguments();
			IF Invoke.bError AND Invoke.nError = E_AdsErr.DEVICE_NOTIFYHNDINVALID THEN
				Invoke.bBusy := TRUE;
				Invoke.bError := FALSE;
				Invoke.nError := E_AdsErr.NOERR;
				eStep := HNDBYNAME;
			END_IF
		END_IF
END_CASE;
END_METHOD

PROPERTY PROTECTED nAmsPort : Tc2_System.T_AmsPort
GET
nAmsPort := nAmsPortField;
END_GET
SET
nAmsPortField := nAmsPort;
END_SET
END_PROPERTY

METHOD NoReturnValue : I_RpcInvoke
NoReturnValue := THIS^;
END_METHOD

METHOD PRIVATE ReadValueByHandle : ST_AdsStatus
VAR_INPUT
	pArgs		: PVOID;
	nLenArgs 	: UDINT;
	pRetVal		: PVOID;
	nLenRetVal 	: UDINT;
END_VAR

VAR
	nNullDummy 	: UDINT;
END_VAR

IF pArgs = NULL THEN
	pArgs := ADR(nNullDummy);
	nLenArgs := 0;
END_IF
	
IF pRetVal = NULL THEN
	pRetVal := ADR(nNullDummy);
	nLenRetVal := 0;
END_IF

fbRdWrReq(
		IDXGRP:= ADSIGRP_SYM_VALBYHND, 
		IDXOFFS:= nSymbolHandle, 
		WRITELEN:=nLenArgs, 
		READLEN:= nLenRetVal , 
		SRCADDR:= pArgs, 
		DESTADDR:= pRetVal, 
		WRTRD:= TRUE, 
		TMOUT:= tAdsTimeOutField, 
		BUSY=> ReadValueByHandle.bBusy, 
		ERR=> ReadValueByHandle.bError, 
		ERRID=> ReadValueByHandle.nError);
END_METHOD

METHOD ReleaseHandle : ST_AdsStatus
IF THIS^.nSymbolHandle = cNoSymbolNameHandle THEN
	RETURN;
END_IF

IF nHandleToRelease = cNoSymbolNameHandle THEN
	fbAdsWrReqRelHandle(WRITE:= FALSE);
	nHandleToRelease := THIS^.nSymbolHandle;
END_IF

fbAdsWrReqRelHandle(
	NETID:= THIS^.sAmsNetIdField, 
	PORT:= THIS^.nAmsPortField, 
	IDXGRP:= ADSIGRP_SYM_RELEASEHND, 
	IDXOFFS:= 16#0, 
	LEN:= SIZEOF(nHandleToRelease), 
	SRCADDR:= ADR(nHandleToRelease), 
	WRITE:= TRUE, 
	TMOUT:= tAdsTimeOutField, 
	BUSY=> ReleaseHandle.bBusy, 
	ERR=> ReleaseHandle.bError, 
	ERRID=> ReleaseHandle.nError);
	
IF NOT fbAdsWrReqRelHandle.BUSY OR fbAdsWrReqRelHandle.ERR THEN
	eStep := HNDBYNAME;
	nHandleToRelease := cNoSymbolNameHandle;	
END_IF
END_METHOD

METHOD Reset
VAR_INPUT
END_VAR
ResetArguments();
ReleaseHandle();
nHandleToRelease := cNoSymbolNameHandle;
fbAdsWrReqRelHandle(WRITE:= FALSE);
fbRdWrReq(WRTRD:= FALSE);
eArgs := NO_LOCK;
END_METHOD

METHOD PRIVATE ResetArguments
VAR_INPUT
END_VAR
fbArguments.Reset();
END_METHOD

METHOD ReturnValue : I_RpcInvoke
VAR_INPUT
	anyRetVal	: ANY;
END_VAR
VAR
	stAny : ST_AnyType;
END_VAR
ReturnValue := THIS^;

IF eArgs = LOCK THEN
	RETURN;
END_IF

IF anyRetVal.diSize <= 0 THEN
	RETURN;
END_IF

stAny := F_ToAnyType(anyRetVal);

fbArguments.SetRetVal(stAny);
END_METHOD

PROPERTY PROTECTED sAmsNetId : Tc2_System.T_AmsNetID
GET
sAmsNetId := sAmsNetIdField;
END_GET
SET
sAmsNetIdField := sAmsNetId;
END_SET
END_PROPERTY

PROPERTY PROTECTED sRpcSymbol : T_MaxString
GET
sRpcSymbol := THIS^.sRpcSymbolField;
END_GET
SET
IF sRpcSymbol <> '' THEN
	sRpcSymbolField := sRpcSymbol;
END_IF
END_SET
END_PROPERTY

PROPERTY tAdsTimeOut : TIME
GET
tAdsTimeOut := tAdsTimeOutField;
END_GET
SET
IF tAdsTimeout > T#0MS THEN
	tAdsTimeOutField := tAdsTimeOut;
END_IF
END_SET
END_PROPERTY

METHOD VarInOut : I_RpcArguments
VAR_INPUT
	anyArg	: ANY;
END_VAR

VAR
	stAny : ST_AnyType;
	eAdsErr : E_AdsErr;
END_VAR
VarInOut := THIS^;

IF eArgs = LOCK THEN
	RETURN;
END_IF

IF anyArg.diSize <= 0 THEN
	RETURN;
END_IF

stAny := F_ToAnyType(anyArg);

eAdsErr := fbArguments.SetVarInOut(stAny);
IF eAdsErr <> E_AdsErr.NOERR THEN
	RETURN;
END_IF
END_METHOD

METHOD VarInput : I_RpcArguments
VAR_INPUT
	anyArg	: ANY;
END_VAR
VAR
	stAny : ST_AnyType;
	eAdsErr : E_AdsErr;
END_VAR
VarInput := THIS^;

IF eArgs = LOCK THEN
	RETURN;
END_IF

stAny := F_ToAnyType(anyArg);

eAdsErr := fbArguments.SetVarInput(stAny);
IF eAdsErr <> E_AdsErr.NOERR THEN
	RETURN;
END_IF
END_METHOD

METHOD VarOutput : I_RpcArguments
VAR_INPUT
	anyArg	: ANY;
END_VAR
VAR
	stAny : ST_AnyType;
	eAdsErr : E_AdsErr;
END_VAR
VarOutput := THIS^;

IF eArgs = LOCK THEN
	RETURN;
END_IF

stAny := F_ToAnyType(anyArg);

eAdsErr := fbArguments.SetVarOutput(stAny);
IF eAdsErr <> E_AdsErr.NOERR THEN
	RETURN;
END_IF
END_METHOD

END_FUNCTION_BLOCK

// ---- POUs/internal/FB_ArgumentsBuffer.TcPOU
{attribute 'no_explicit_call' := 'do not call this POU directly'}
{attribute 'hide_all_locals'}
FUNCTION_BLOCK INTERNAL FINAL FB_ArgumentsBuffer IMPLEMENTS I_ArgsBuffer

VAR
	aVarInputBuffer			: ARRAY [0..cMaxArgsBuffer - 1] OF BYTE;
	nVarInputBufferIndex	: UDINT := 0;
	aVarInputArgs			: ARRAY [0..cMaxArgs - 1] OF ST_AnyType;
	nVarInputIndex			: UDINT := 0;
	
	aVarInOutBuffer			: ARRAY [0..cMaxArgsBuffer - 1] OF BYTE;
	nVarInOutBufferIndex	: UDINT := 0;
	aAnyVarInOut			: ARRAY [0..cMaxArgs - 1] OF ST_AnyType;
	nAnyVarInOutIndex		: UDINT := 0;
	
	nRetValSizeTotal		: UDINT := 0;						// total size in Bytes of all In/Out arguments + return value
	stAnyRetVal				: ST_AnyType;
	
END_VAR

VAR CONSTANT
	cMaxArgsBuffer		: UDINT := Param_Args.cMaxArgsBuffer;	// max sizeof aArgs buffer array.
	cMaxArgs			: USINT := Param_Args.cMaxArgs;			// max length method arguments
END_VAR

METHOD GetRetVal : E_AdsErr
VAR_INPUT
END_VAR
VAR 
	i : UDINT;
	nLen : UDINT;
	pPtr : POINTER TO PVOID;
END_VAR
nVarInOutBufferIndex := 0;

IF stAnyRetVal.pValue <> NULL THEN
	nLen := TO_UDINT(stAnyRetVal.nSize);
	IF nLen > SIZEOF(aVarInOutBuffer) THEN
		GetRetVal := E_AdsErr.DEVICE_NOMEMORY;
		RETURN;
	END_IF
	MEMCPY(destAddr:= stAnyRetVal.pValue, srcAddr:= ADR(aVarInOutBuffer), n:= nLen);
	nVarInOutBufferIndex := nVarInOutBufferIndex + nLen;
END_IF


FOR i:=0 TO nAnyVarInOutIndex DO
	nLen := TO_UDINT(aAnyVarInOut[i].nSize);
	IF nLen + nVarInOutBufferIndex > SIZEOF(aVarInOutBuffer) THEN
		GetRetVal := E_AdsErr.DEVICE_NOMEMORY;
		RETURN;
	END_IF	
	IF aAnyVarInOut[i].TypeClass = __SYSTEM.TYPE_CLASS.TYPE_POINTER THEN
		pPtr := aAnyVarInOut[i].pValue;
		MEMCPY(destAddr:= pPtr^, srcAddr:= ADR(aVarInOutBuffer[nVarInOutBufferIndex]), n:= nLen);
	ELSE
		MEMCPY(destAddr:= aAnyVarInOut[i].pValue, srcAddr:= ADR(aVarInOutBuffer[nVarInOutBufferIndex]), n:= nLen);
	END_IF
	nVarInOutBufferIndex := nVarInOutBufferIndex + nLen;
END_FOR
END_METHOD

PROPERTY nArgsLength : UDINT
GET
nArgsLength := THIS^.nVarInputBufferIndex;
END_GET
END_PROPERTY

PROPERTY nRetValLength : UDINT
GET
nRetValLength := THIS^.nRetValSizeTotal;
END_GET
END_PROPERTY

PROPERTY pArgsBuffer : POINTER TO BYTE
GET
pArgsBuffer := ADR(aVarInputBuffer);
END_GET
END_PROPERTY

PROPERTY pRetValBuffer : POINTER TO BYTE
GET
pRetValBuffer := ADR(aVarInOutBuffer);
END_GET
END_PROPERTY

METHOD Reset
MEMSET(ADR(aVarInputBuffer), 16#0, SIZEOF(aVarInputBuffer));
MEMSET(ADR(aVarInputArgs), 16#0, SIZEOF(aVarInputArgs));
MEMSET(ADR(aVarInOutBuffer), 16#0, SIZEOF(aVarInOutBuffer));
MEMSET(ADR(aAnyVarInOut), 16#0, SIZEOF(aAnyVarInOut));
MEMSET(ADR(stAnyRetVal), 16#0, SIZEOF(stAnyRetVal));
nVarInputIndex := 0;
nVarInputBufferIndex := 0;
nVarInputBufferIndex := 0;
nAnyVarInOutIndex := 0;
nRetValSizeTotal := 0;
END_METHOD

METHOD SetRetVal
VAR_INPUT
	stAny : ST_AnyType;
END_VAR

stAnyRetVal := stAny;
nRetValSizeTotal := nRetValSizeTotal + TO_UDINT(stAny.nSize);
END_METHOD

METHOD SetVarInOut : E_AdsErr
VAR_INPUT
	stAny : ST_AnyType;
END_VAR
VAR
	eAdsErr : E_AdsErr;
END_VAR
IF stAny.pValue = NULL OR stAny.nSize <= 0 THEN
	SetVarInOut := E_AdsErr.DEVICE_INVALIDPARM;
	RETURN;
END_IF
IF nVarInOutBufferIndex + TO_UDINT(stAny.nSize) > SIZEOF(aVarInOutBuffer) THEN
	SetVarInOut := E_AdsErr.DEVICE_NOMEMORY;
	RETURN;
END_IF
IF nAnyVarInOutIndex > cMaxArgs -1  THEN
	SetVarInOut := E_AdsErr.DEVICE_NOMEMORY;
	RETURN;
END_IF

eAdsErr := SetVarInput(stAny);
IF eAdsErr <> E_AdsErr.NOERR THEN
	RETURN;
END_IF


aAnyVarInOut[nAnyVarInOutIndex] := stAny;
nAnyVarInOutIndex := nAnyVarInOutIndex + 1;
nRetValSizeTotal := nRetValSizeTotal + TO_UDINT(stAny.nSize);
END_METHOD

METHOD SetVarInput : E_AdsErr
VAR_INPUT
	stAny : ST_AnyType;
END_VAR
IF nVarInputBufferIndex + TO_UDINT(stAny.nSize) > SIZEOF(aVarInputBuffer) THEN
	SetVarInput := E_AdsErr.DEVICE_NOMEMORY;
	RETURN;
END_IF
IF nVarInputIndex > cMaxArgs -1  THEN
	SetVarInput := E_AdsErr.DEVICE_NOMEMORY;
	RETURN;
END_IF

aVarInputArgs[nVarInputIndex] := stAny;
nVarInputIndex := nVarInputIndex + 1;

MEMCPY(ADR(aVarInputBuffer[nVarInputBufferIndex]), stAny.pValue , TO_UDINT(stAny.nSize));
nVarInputBufferIndex := nVarInputBufferIndex + TO_UDINT(stAny.nSize);
END_METHOD

METHOD SetVarOutput : E_AdsErr
VAR_INPUT
	stAny : ST_AnyType;
END_VAR

IF stAny.pValue = NULL OR stAny.nSize <= 0 THEN
	SetVarOutput := E_AdsErr.DEVICE_INVALIDPARM;
	RETURN;
END_IF
IF nVarInOutBufferIndex + TO_UDINT(stAny.nSize) > SIZEOF(aVarInOutBuffer) THEN
	SetVarOutput := E_AdsErr.DEVICE_NOMEMORY;
	RETURN;
END_IF
IF nAnyVarInOutIndex > cMaxArgs -1  THEN
	SetVarOutput := E_AdsErr.DEVICE_NOMEMORY;
	RETURN;
END_IF


aAnyVarInOut[nAnyVarInOutIndex] := stAny;
nAnyVarInOutIndex := nAnyVarInOutIndex + 1;
nRetValSizeTotal := nRetValSizeTotal + TO_UDINT(stAny.nSize);
END_METHOD

END_FUNCTION_BLOCK

// ---- POUs/F_ToAnyType.TcPOU
FUNCTION F_ToAnyType : ST_AnyType
VAR_INPUT
	anyArg	: ANY;
END_VAR

F_ToAnyType.pValue := anyArg.pValue;
F_ToAnyType.nSize := anyArg.diSize;
F_ToAnyType.TypeClass := anyArg.TypeClass;

END_FUNCTION

// ---- TESTs/FB_RPC_Dynamic_Tests.TcPOU
{attribute 'reflection'}
FUNCTION_BLOCK INTERNAL FINAL FB_RPC_Dynamic_Tests EXTENDS TcUnit.FB_TestSuite
VAR
	{attribute 'instance-path'} 
    {attribute 'noinit'} 
	sTestName			: T_MaxString;
	sActiveStep			: T_MaxString;
	nSequence			: INT;
	nSeqOld				: INT;
	nRpcMethodInvoked 	: UDINT;
	aSUTs				: ARRAY[0..255] OF I_RpcReleaseHandle;
END_VAR
VAR_TEMP
	eMode	: E_Mode;
END_VAR

CASE nSequence OF
	0:
		TEST(sTestName);
		F_IncrementStep(nStepToInc:= nSequence, sActiveStep:= sActiveStep, eMode:= E_Mode.INC);
	1:
		sActiveStep := 'ShouldInvokeMethod_NoArguments_NoReturnValue_Successfully';
		TEST(sActiveStep);
		eMode := ShouldInvokeMethod_NoArguments_NoReturnValue_Successfully();
		F_IncrementStep(nStepToInc:= nSequence, sActiveStep, eMode);
	2:
		sActiveStep := 'ShouldInvokeMethod_NoArguments_ReturnValueBoolean_Successfully';
		TEST(sActiveStep);
		eMode := ShouldInvokeMethod_NoArguments_ReturnValueBoolean_Successfully();
		F_IncrementStep(nStepToInc:= nSequence, sActiveStep, eMode);
	3:	
		sActiveStep := 'ShouldInvokeMethod_OneArgument_NoReturnValue_Successfully';
		TEST(sActiveStep);
		eMode := ShouldInvokeMethod_OneArgument_NoReturnValue_Successfully();
		F_IncrementStep(nStepToInc:= nSequence, sActiveStep, eMode);	
	4:	
		sActiveStep := 'ShouldInvokeMethod_OneArgument_NoReturnValue_Successfully';
		TEST(sActiveStep);
		eMode := ShouldInvokeMethod_OneArgument_NoReturnValue_Successfully();
		F_IncrementStep(nStepToInc:= nSequence, sActiveStep, eMode);	
	5:	
		sActiveStep := 'ShouldInvokeMethod_TwoArguments_ReturnValue_Successfully';
		TEST(sActiveStep);
		eMode := ShouldInvokeMethod_TwoArguments_ReturnValue_Successfully();
		F_IncrementStep(nStepToInc:= nSequence, sActiveStep, eMode);
	6:	
		sActiveStep := 'ShouldInvokeMethod_ThreeArguments_ReturnValue_Successfully';
		TEST(sActiveStep);
		eMode := ShouldInvokeMethod_ThreeArguments_ReturnValue_Successfully();
		F_IncrementStep(nStepToInc:= nSequence, sActiveStep, eMode);		
	7:	
		sActiveStep := 'ShouldInvokeMethod_VarInOutConstant_ReturnValue_Successfully';
		TEST(sActiveStep);
		eMode := ShouldInvokeMethod_VarInOutConstant_ReturnValue_Successfully();
		F_IncrementStep(nStepToInc:= nSequence, sActiveStep, eMode);	
	8:	
		sActiveStep := 'ShouldInvokeMethod_VarOutput_ReturnValue_Successfully';
		TEST(sActiveStep);
		eMode := ShouldInvokeMethod_VarOutput_ReturnValue_Successfully();
		F_IncrementStep(nStepToInc:= nSequence, sActiveStep, eMode);	
	9:	
		sActiveStep := 'ShouldInvokeMethod_TwoVarOutput_ReturnValue_Successfully';
		TEST(sActiveStep);
		eMode := ShouldInvokeMethod_TwoVarOutput_ReturnValue_Successfully();
		F_IncrementStep(nStepToInc:= nSequence, sActiveStep, eMode);	
	10:	
		sActiveStep := 'ShouldInvokeMethod_VarInput_VarInOut_VarOutput_ReturnValue_Successfully';
		TEST(sActiveStep);
		eMode := ShouldInvokeMethod_VarInput_VarInOut_VarOutput_ReturnValue_Successfully();
		F_IncrementStep(nStepToInc:= nSequence, sActiveStep, eMode);		
	11: 
		sActiveStep := 'ShouldReturnError0x705';
		TEST(sActiveStep);
		eMode := ShouldReturnError0x705();
		F_IncrementStep(nStepToInc:= nSequence, sActiveStep, eMode);	
	12: 
		sActiveStep := 'ShouldReturnError0x710';
		TEST(sActiveStep);
		eMode := ShouldReturnError0x710();
		F_IncrementStep(nStepToInc:= nSequence, sActiveStep, eMode);	
	13: 
		sActiveStep := 'ShouldReleaseAllSymbolHandleSuccessfully';
		TEST(sActiveStep);
		eMode := ShouldReleaseAllSymbolHandleSuccessfully();
		F_IncrementStep(nStepToInc:= nSequence, sActiveStep, eMode);	
	ELSE
		TEST_FINISHED_NAMED(sTestName);
END_CASE

IF nSequence <> nSeqOld THEN
	nRpcMethodInvoked := 0;
	nSeqOld := nSequence;
END_IF;

{attribute 'TcRpcEnable'}
METHOD NoParameter_NoReturnValue

nRpcMethodInvoked := nRpcMethodInvoked + 1;
END_METHOD

{attribute 'TcRpcEnable'}
METHOD NoParameter_ReturnValue : BOOL
VAR_INPUT
END_VAR
nRpcMethodInvoked := nRpcMethodInvoked + 1;
NoParameter_ReturnValue := nRpcMethodInvoked > 0;
END_METHOD

{attribute 'TcRpcEnable'}
METHOD OneParameter_NoReturnValue
VAR_INPUT
	nArg1 	: UDINT;
END_VAR
nRpcMethodInvoked := nArg1;
END_METHOD

METHOD Register
VAR_INPUT
	ipRpcReleaseHandle	: I_RpcReleaseHandle;
END_VAR

VAR
	i :UINT;
END_VAR


FOR i:=0 TO 255 DO	
	IF aSUTs[i] = ipRpcReleaseHandle THEN
		EXIT;
	END_IF
	IF aSUTs[i] <> NULL THEN
		CONTINUE;
	END_IF
	
	aSUTs[i] := ipRpcReleaseHandle;
	EXIT;
END_FOR
END_METHOD

METHOD ShouldInvokeMethod_NoArguments_NoReturnValue_Successfully : E_Mode

VAR_INST
	fbSUT		: FB_RPC_Dynamic;
END_VAR

VAR
	stRetVal	: ST_AdsStatus;
	eMode		: E_Mode := E_MODE.BUSY;
END_VAR
// Arrange
Register(fbSUT);
fbSUT.Configure()
	.WithAmsNetId(GCL.cLocalAmsNetId)
	.WithAmsPort(_AppInfo.AdsPort)
	.WithSymbolPath('PRG_UnitTests.fbRpcDynamicTests','NoParameter_NoReturnValue')
	.Build();

// Act
stRetVal := fbSUT.Invoke();

IF NOT stRetVal.bBusy THEN
	eMode := E_Mode.INC;
	
	// Assert
	AssertFalse(Condition:= stRetVal.bError, Message:= 'Expected method NoParameter_NoReturnValue to return no error.');
	AssertEquals_UDINT(Expected:= E_AdsErr.NOERR, Actual:= stRetVal.nError, Message:= 'Expected method NoParameter_NoReturnValue to return no error.');
	AssertEquals_UDINT(Expected:= 1, Actual:= nRpcMethodInvoked, Message:= 'Expected method NoParameter_NoReturnValue to be invoked once.');
END_IF

ShouldInvokeMethod_NoArguments_NoReturnValue_Successfully := eMode;
END_METHOD

METHOD ShouldInvokeMethod_NoArguments_ReturnValueBoolean_Successfully : E_Mode

VAR_INST
	fbSUT		: FB_RPC_Dynamic;
END_VAR

VAR
	stRetVal	: ST_AdsStatus;
	eMode		: E_Mode := E_MODE.BUSY;
	bActual		: BOOL;
END_VAR
// Arrange
Register(fbSUT);
fbSUT.Configure()
	.WithAmsNetId(GCL.cLocalAmsNetId)
	.WithAmsPort(_AppInfo.AdsPort)
	.WithSymbolPath('PRG_UnitTests.fbRpcDynamicTests','NoParameter_ReturnValue')
	.Build();
	
// Act
stRetVal := fbSUT.ReturnValue(bActual).Invoke();

IF NOT stRetVal.bBusy THEN
	eMode := E_Mode.INC;
	// Assert
	AssertFalse(Condition:= stRetVal.bError, Message:= 'Expected method NoParameter_ReturnValue to return no error.');
	AssertEquals_UDINT(Expected:= E_AdsErr.NOERR, Actual:= stRetVal.nError, Message:= 'Expected method NoParameter_ReturnValue to return no error.');
	AssertEquals_UDINT(Expected:= 1, Actual:= nRpcMethodInvoked, Message:= 'Expected method NoParameter_ReturnValue to be invoked once.');
	AssertTrue(Condition:= bActual, Message:= 'Expected method NoParameter_ReturnValue to return TRUE.');
END_IF

ShouldInvokeMethod_NoArguments_ReturnValueBoolean_Successfully := eMode;
END_METHOD

METHOD ShouldInvokeMethod_OneArgument_NoReturnValue_Successfully : E_Mode

VAR_INST
	fbSUT		: FB_RPC_Dynamic;
END_VAR

VAR
	stRetVal	: ST_AdsStatus;
	eMode		: E_Mode := E_MODE.BUSY;
	nArg		: UDINT;
END_VAR
// Arrange
Register(fbSUT);
fbSUT.Configure()
	.WithAmsNetId(GCL.cLocalAmsNetId)
	.WithAmsPort(_AppInfo.AdsPort)
	.WithSymbolPath('PRG_UnitTests.fbRpcDynamicTests','OneParameter_NoReturnValue')
	.Build();

nArg := 123;

// Act
stRetVal := fbSUT.VarInput(nArg).NoReturnValue().Invoke();

IF NOT stRetVal.bBusy THEN
	eMode := E_Mode.INC;
	
	// Assert
	AssertFalse(Condition:= stRetVal.bError, Message:= 'Expected method OneParameter_NoReturnValue to return no error.');
	AssertEquals_UDINT(Expected:= E_AdsErr.NOERR, Actual:= stRetVal.nError, Message:= 'Expected method OneParameter_NoReturnValue to return no error.');
	AssertEquals_UDINT(Expected:= nArg, Actual:= nRpcMethodInvoked, Message:= 'Expected method OneParameter_NoReturnValue to be invoked with value 123.');
END_IF

ShouldInvokeMethod_OneArgument_NoReturnValue_Successfully := eMode;
END_METHOD

METHOD ShouldInvokeMethod_ThreeArguments_ReturnValue_Successfully : E_Mode

VAR_INST
	fbSUT		: FB_RPC_Dynamic;
END_VAR

VAR
	stRetVal	: ST_AdsStatus;
	eMode		: E_Mode := E_MODE.BUSY;
	nArg1		: UDINT;
	stArg2		: ST_AdsStatus;	// IN_OUT!
	sArg3		: STRING;
	sActualRetVal : STRING;
END_VAR
// Arrange
Register(fbSUT);
fbSUT.Configure()
	.WithAmsNetId(GCL.cLocalAmsNetId)
	.WithAmsPort(_AppInfo.AdsPort)
	.WithSymbolPath('PRG_UnitTests.fbRpcDynamicTests','ThreeParameters_ReturnValue')
	.Build();

nArg1 := 456;
stArg2.bBusy := FALSE;
stArg2.bError := TRUE;
stArg2.nError := 321;
sArg3 := 'third Argument';

// Act
stRetVal := fbSUT.VarInput(nArg1).VarInOut(stArg2).VarInput(sArg3).ReturnValue(sActualRetVal).Invoke();

IF NOT stRetVal.bBusy THEN
	eMode := E_Mode.INC;
	
	// Assert
	AssertFalse(Condition:= stRetVal.bError, Message:= 'Expected method TwoParameters_ReturnValue to return no error.');
	AssertEquals_UDINT(Expected:= E_AdsErr.NOERR, Actual:= stRetVal.nError, Message:= 'Expected method ThreeParameters_ReturnValue to return no error.');
	AssertEquals_UDINT(Expected:= nArg1, Actual:= nRpcMethodInvoked, Message:= 'Expected method ThreeParameters_ReturnValue to be invoked with value 456.');
	AssertTrue(Condition:= stArg2.bBusy, Message:= 'Expected method ThreeParameters_ReturnValue to invert bBusy of VAR_IN_OUT');
	AssertFalse(Condition:= stArg2.bError, Message:= 'Expected method ThreeParameters_ReturnValue to invert bError of VAR_IN_OUT');
	AssertEquals_UDINT(Expected:= 321 * 2, Actual:= stArg2.nError, Message:= 'Expected method ThreeParameters_ReturnValue to double value nError of VAR_IN_OUT');
	AssertEquals_STRING(Expected:= sArg3, Actual:= sActualRetVal, Message:= 'Expected method ThreeParameters_ReturnValue to return value .');
END_IF

ShouldInvokeMethod_ThreeArguments_ReturnValue_Successfully := eMode;
END_METHOD

METHOD ShouldInvokeMethod_TwoArguments_ReturnValue_Successfully : E_Mode

VAR_INST
	fbSUT		: FB_RPC_Dynamic;
END_VAR

VAR
	stRetVal	: ST_AdsStatus;
	eMode		: E_Mode := E_MODE.BUSY;
	nArg1		: UDINT;
	sArg2		: STRING;
	sActualRetVal : STRING;
END_VAR
// Arrange
Register(fbSUT);
fbSUT.Configure()
	.WithAmsNetId(GCL.cLocalAmsNetId)
	.WithAmsPort(_AppInfo.AdsPort)
	.WithSymbolPath('PRG_UnitTests.fbRpcDynamicTests','TwoParameters_ReturnValue')
	.Build();
	
nArg1 := 456;
sArg2 := 'second Argument';

// Act
stRetVal := fbSUT.VarInput(nArg1).VarInput(sArg2).ReturnValue(sActualRetVal).Invoke();

IF NOT stRetVal.bBusy THEN
	eMode := E_Mode.INC;
	
	// Assert
	AssertFalse(Condition:= stRetVal.bError, Message:= 'Expected method TwoParameters_ReturnValue to return no error.');
	AssertEquals_UDINT(Expected:= E_AdsErr.NOERR, Actual:= stRetVal.nError, Message:= 'Expected method TwoParameters_ReturnValue to return no error.');
	AssertEquals_UDINT(Expected:= nArg1, Actual:= nRpcMethodInvoked, Message:= 'Expected method TwoParameters_ReturnValue to be invoked with value 456.');
	AssertEquals_STRING(Expected:= sArg2, Actual:= sActualRetVal, Message:= 'Expected method TwoParameters_ReturnValue to return value .');
END_IF

ShouldInvokeMethod_TwoArguments_ReturnValue_Successfully := eMode;
END_METHOD

METHOD ShouldInvokeMethod_TwoVarOutput_ReturnValue_Successfully : E_Mode

VAR_INST
	fbSUT		: FB_RPC_Dynamic;
END_VAR

VAR
	stRetVal	: ST_AdsStatus;
	eMode		: E_Mode := E_MODE.BUSY;
	stArg		: ST_AdsStatus;
	nA			: UDINT;
	nActualRetVal : UDINT;
END_VAR
// Arrange
Register(fbSUT);
fbSUT.Configure()
	.WithAmsNetId(GCL.cLocalAmsNetId)
	.WithAmsPort(_AppInfo.AdsPort)
	.WithSymbolPath('PRG_UnitTests.fbRpcDynamicTests','TwoVarOutput_ReturnValue')
	.Build();
	
// Act
stRetVal := fbSUT.VarOutput(stArg).VarOutput(nA).ReturnValue(nActualRetVal).Invoke();

IF NOT stRetVal.bBusy THEN
	eMode := E_Mode.INC;
	
	// Assert
	AssertFalse(Condition:= stRetVal.bError, Message:= 'Expected method VarOutput_ReturnValue to return no error.');
	AssertEquals_UDINT(Expected:= E_AdsErr.NOERR, Actual:= stRetVal.nError, Message:= 'Expected method VarOutput_ReturnValue to return no error.');
	AssertFalse(Condition:= stArg.bBusy, Message:= 'Expected method VarOutput_ReturnValue to return stArg.bBusy = FALSE');
	AssertTrue(Condition:= stArg.bError, Message:= 'Expected method VarOutput_ReturnValue to return stArg.bError = TRUE');
	AssertEquals_UDINT(Expected:= 123, Actual:= stARg.nError, Message:= 'Expected method VarOutput_ReturnValue to return stArg.nError = 123');
	AssertEquals_UDINT(Expected:= 789, Actual:= nA, Message:= 'Expected method VarOutput_ReturnValue to return nA = 789');
	AssertEquals_UDINT(Expected:= 456, Actual:= nActualRetVal, Message:= 'Expected method VarOutput_ReturnValue to return 456.');
END_IF

ShouldInvokeMethod_TwoVarOutput_ReturnValue_Successfully := eMode;
END_METHOD

METHOD ShouldInvokeMethod_VarInOutConstant_ReturnValue_Successfully : E_Mode

VAR_INST
	fbSUT		: FB_RPC_Dynamic;
END_VAR

VAR
	stRetVal	: ST_AdsStatus;
	eMode		: E_Mode := E_MODE.BUSY;
	stArg		: ST_LibVersion;
	nActualRetVal : UDINT;
END_VAR
// Arrange
Register(fbSUT);
fbSUT.Configure()
	.WithAmsNetId(GCL.cLocalAmsNetId)
	.WithAmsPort(_AppInfo.AdsPort)
	.WithSymbolPath('PRG_UnitTests.fbRpcDynamicTests','VarInOutConstant_ReturnValue')
	.Build();
	
stArg.nFlags := 987;

// Act
stRetVal := fbSUT.VarInOut(stArg).ReturnValue(nActualRetVal).Invoke();

IF NOT stRetVal.bBusy THEN
	eMode := E_Mode.INC;
	
	// Assert
	AssertFalse(Condition:= stRetVal.bError, Message:= 'Expected method VarInOutConstant_ReturnValue to return no error.');
	AssertEquals_UDINT(Expected:= E_AdsErr.NOERR, Actual:= stRetVal.nError, Message:= 'Expected method VarInOutConstant_ReturnValue to return no error.');
	AssertEquals_DWORD(Expected:= 987, Actual:= stArg.nFlags, Message:= 'Expected method VarInOutConstant_ReturnValue to be invoked with value 987.');
	AssertEquals_UDINT(Expected:= 987, Actual:= nActualRetVal, Message:= 'Expected method VarInOutConstant_ReturnValue to be invoked with value 987.');
END_IF

ShouldInvokeMethod_VarInOutConstant_ReturnValue_Successfully := eMode;
END_METHOD

METHOD ShouldInvokeMethod_VarInput_VarInOut_VarOutput_ReturnValue_Successfully : E_Mode

VAR_INST
	fbSUT		: FB_RPC_Dynamic;
END_VAR

VAR
	stRetVal	: ST_AdsStatus;
	eMode		: E_Mode := E_MODE.BUSY;
		
	sStrIn		: STRING;
	nIn			: INT;
	nInOut 		: INT;
	stArgOut	: ST_AdsStatus;
	sStrOut		: STRING;	
	sRetVal		: STRING;
END_VAR
// Arrange
Register(fbSUT);
fbSUT.Configure()
	.WithAmsNetId(GCL.cLocalAmsNetId)
	.WithAmsPort(_AppInfo.AdsPort)
	.WithSymbolPath('PRG_UnitTests.fbRpcDynamicTests','VarInput_VarInOut_VarOutput_ReturnValue')
	.Build();
	
sStrIn	:= 'Input String';
nIn		:= -666;
nInOut	:= 777;

// Act
stRetVal := fbSUT.VarInput(sStrIn).VarInput(nIn).VarInOut(nInOut).VarOutput(stArgOut).VarOutput(sStrOut).ReturnValue(sRetVal).Invoke();

IF NOT stRetVal.bBusy THEN
	eMode := E_Mode.INC;
	
	// Assert
	AssertFalse(Condition:= stRetVal.bError, Message:= 'Expected method VarInput_VarInOut_VarOutput_ReturnValue to return no error.');
	AssertEquals_UDINT(Expected:= E_AdsErr.NOERR, Actual:= stRetVal.nError, Message:= 'Expected method VarInput_VarInOut_VarOutput_ReturnValue to return no error.');
	AssertTrue(Condition:= stArgOut.bBusy, Message:= 'Expected method VarInput_VarInOut_VarOutput_ReturnValue to return stArgOut.bBusy = TRUE');
	AssertFalse(Condition:= stArgOut.bError, Message:= 'Expected method VarInput_VarInOut_VarOutput_ReturnValue to return stArgOut.bError = FALSE');
	AssertEquals_UDINT(Expected:= 222, Actual:= stArgOut.nError, Message:= 'Expected method VarInput_VarInOut_VarOutput_ReturnValue to return stArgOut.nError = 222');
	AssertEquals_STRING(Expected:= 'sStrOut: Input String', Actual:= sStrOut,
						Message:= 'Expected method VarInput_VarInOut_VarOutput_ReturnValue to return "sStrOut: Input String"');
	AssertEquals_STRING(Expected:= 'ReturnValue: Input String', Actual:= sRetVal,
						Message:= 'Expected method VarInput_VarInOut_VarOutput_ReturnValue to return "ReturnValue: Input String"');
END_IF

ShouldInvokeMethod_VarInput_VarInOut_VarOutput_ReturnValue_Successfully := eMode;
END_METHOD

METHOD ShouldInvokeMethod_VarOutput_ReturnValue_Successfully : E_Mode

VAR_INST
	fbSUT		: FB_RPC_Dynamic;
END_VAR

VAR
	stRetVal	: ST_AdsStatus;
	eMode		: E_Mode := E_MODE.BUSY;
	stArg		: ST_AdsStatus;
	nActualRetVal : UDINT;
END_VAR
// Arrange
Register(fbSUT);
fbSUT.Configure()
	.WithAmsNetId(GCL.cLocalAmsNetId)
	.WithAmsPort(_AppInfo.AdsPort)
	.WithSymbolPath('PRG_UnitTests.fbRpcDynamicTests','VarOutput_ReturnValue')
	.Build();

// Act
stRetVal := fbSUT.VarOutput(stArg).ReturnValue(nActualRetVal).Invoke();

IF NOT stRetVal.bBusy THEN
	eMode := E_Mode.INC;
	
	// Assert
	AssertFalse(Condition:= stRetVal.bError, Message:= 'Expected method VarOutput_ReturnValue to return no error.');
	AssertEquals_UDINT(Expected:= E_AdsErr.NOERR, Actual:= stRetVal.nError, Message:= 'Expected method VarOutput_ReturnValue to return no error.');
	AssertTrue(Condition:= stArg.bBusy, Message:= 'Expected method VarOutput_ReturnValue to return bBusy = TRUE.');
	AssertFalse(Condition:= stArg.bError, Message:= 'Expected method VarOutput_ReturnValue to return bError = FALSE');
	AssertEquals_UDINT(Expected:= 456, Actual:= stARg.nError, Message:= 'Expected method VarOutput_ReturnValue to return VAR_OUTPUT 456.');
	AssertEquals_UDINT(Expected:= 123, Actual:= nActualRetVal, Message:= 'Expected method VarOutput_ReturnValue to return 123.');
END_IF

ShouldInvokeMethod_VarOutput_ReturnValue_Successfully := eMode;
END_METHOD

METHOD ShouldReleaseAllSymbolHandleSuccessfully : E_Mode

VAR
	stRetVal	: ST_AdsStatus;
	ipSUT		: I_RpcReleaseHandle;
END_VAR

VAR_INST
	nIndex 		: UINT := 0;
END_VAR


ipSUT := aSUTs[nIndex];
IF ipSUT = NULL THEN
	ShouldReleaseAllSymbolHandleSuccessfully := E_Mode.INC;
	RETURN;
END_IF

// Act
stRetVal := ipSUT.ReleaseHandle();

IF NOT stRetVal.bBusy THEN
	nIndex := nIndex + 1;	
	// Assert
	AssertFalse(Condition:= stRetVal.bError, Message:= 'Expected ReleaseHandle to return no error.');
	AssertEquals_UDINT(Expected:= E_AdsErr.NOERR, Actual:= stRetVal.nError, Message:= 'Expected ReleaseHandle to return no error.');
END_IF

ShouldReleaseAllSymbolHandleSuccessfully := E_Mode.BUSY;
END_METHOD

METHOD ShouldReturnError0x705 : E_Mode

VAR_INST
	fbSUT		: FB_RPC_Dynamic;
END_VAR

VAR
	stRetVal	: ST_AdsStatus;
	eMode		: E_Mode := E_MODE.BUSY;
	nDummy		: INT;
END_VAR
//Arrange
fbSUT.Configure()
	.WithAmsNetId(GCL.cLocalAmsNetId)
	.WithAmsPort(_AppInfo.AdsPort)
	.WithSymbolPath('PRG_UnitTests.fbRpcDynamicTests','NoParameter_NoReturnValue')
	.Build();

// Act
stRetVal := fbSUT.VarInput(nDummy).NoReturnValue().Invoke();

IF NOT stRetVal.bBusy THEN
	eMode := E_Mode.INC;
	
	// Assert
	AssertTrue(Condition:= stRetVal.bError, Message:= 'Expected method NoParameter_NoReturnValue to return error.');
	AssertEquals_UDINT(Expected:= E_AdsErr.DEVICE_INVALIDSIZE, Actual:= stRetVal.nError, Message:= 'Expected method NoParameter_NoReturnValue to return error ADSERR_DEVICE_INVALIDSIZE.');
	AssertEquals_UDINT(Expected:= 0, Actual:= nRpcMethodInvoked, Message:= 'Expected method NoParameter_NoReturnValue to not be invoked.');
END_IF

ShouldReturnError0x705 := eMode;
END_METHOD

METHOD ShouldReturnError0x710 : E_Mode

VAR_INST
	fbSUT		: FB_RPC_Dynamic;
END_VAR

VAR
	stRetVal	: ST_AdsStatus;
	eMode		: E_Mode := E_MODE.BUSY;
	nDummy		: INT;
END_VAR
// Arrange
fbSUT.Configure()
	.WithAmsNetId(GCL.cLocalAmsNetId)
	.WithAmsPort(_AppInfo.AdsPort)
	.WithSymbolPath('PRG_UnitTests.fbRpcDynamicTests','NotExistingSymbol')
	.Build();

// Act
stRetVal := fbSUT.VarInput(nDummy).NoReturnValue().Invoke();

IF NOT stRetVal.bBusy THEN
	eMode := E_Mode.INC;
	
	// Assert
	AssertTrue(Condition:= stRetVal.bError, Message:= 'Expected return error.');
	AssertEquals_UDINT(Expected:= E_AdsErr.DEVICE_SYMBOLNOTFOUND, Actual:= stRetVal.nError, Message:= 'Expected error ADSERR_DEVICE_SYMBOLNOTFOUND.');
END_IF

ShouldReturnError0x710 := eMode;
END_METHOD

{attribute 'TcRpcEnable'}
METHOD ThreeParameters_ReturnValue : STRING
VAR_INPUT
	nArg1 	: UDINT;
END_VAR
VAR_IN_OUT
	stArg2  : ST_AdsStatus;
END_VAR
VAR_INPUT
	sArg3	: STRING;
END_VAR
nRpcMethodInvoked := nArg1;
stArg2.bBusy := NOT stArg2.bBusy;
stArg2.bError := NOT stARg2.bError;
stARg2.nError := stARg2.nError * 2;
ThreeParameters_ReturnValue := sArg3;
END_METHOD

{attribute 'TcRpcEnable'}
METHOD TwoParameters_ReturnValue : STRING
VAR_INPUT
	nArg1 	: UDINT;
	sArg2	: STRING;
END_VAR
nRpcMethodInvoked := nArg1;
TwoParameters_ReturnValue := sArg2;
END_METHOD

{attribute 'TcRpcEnable'}
METHOD TwoVarOutput_ReturnValue : UDINT
VAR_OUTPUT
	stArg	: ST_AdsStatus;
	nA		: UDINT;
END_VAR

stArg.bBusy := FALSE;
stArg.bError := TRUE;
stArg.nError := 123;
nA := 789;
TwoVarOutput_ReturnValue := 456;
END_METHOD

{attribute 'TcRpcEnable'}
METHOD VarInOutConstant_ReturnValue : DWORD
VAR_IN_OUT CONSTANT
	stArg  : ST_LibVersion;
END_VAR
VarInOutConstant_ReturnValue := stArg.nFlags;
END_METHOD

{attribute 'TcRpcEnable'}
METHOD VarInput_VarInOut_VarOutput_ReturnValue : STRING
VAR_INPUT
	sStrIn	: STRING;
	nIn		: INT;
END_VAR
VAR_IN_OUT
	nInOut	: INT;	
END_VAR
VAR_OUTPUT
	stArgOut	: ST_AdsStatus;
	sStrOut 	: STRING;
END_VAR



nInOut := nInOut + nIn;

stArgOut.bBusy := TRUE;
stArgOut.bError := FALSE;
stArgOut.nError := 222;

sStrOut := CONCAT('sStrOut: ',sStrIn);

VarInput_VarInOut_VarOutput_ReturnValue := CONCAT('ReturnValue: ',sStrIn);
END_METHOD

{attribute 'TcRpcEnable'}
METHOD VarOutput_ReturnValue : UDINT
VAR_OUTPUT
	stArg  : ST_AdsStatus;
END_VAR

stArg.bBusy := TRUE;
stArg.bError := FALSE;
stArg.nError := 456;
VarOutput_ReturnValue := 123;
END_METHOD

END_FUNCTION_BLOCK

// ---- POUs/FB_RPC_Dynamic.TcPOU
{attribute 'no_explicit_call' := 'do not call this POU directly'}
{attribute 'conditionalshow_all_locals'}
// Function Block to invoke RPC calls.
FUNCTION_BLOCK FINAL FB_RPC_Dynamic EXTENDS FB_RpcBase IMPLEMENTS I_RpcDynamicConfig

VAR
	{attribute 'hide'}	
	fbConfig				: FB_RpcConfig;
END_VAR

METHOD INTERNAL ConfigDoneCallback : HRESULT
VAR_INPUT CONSTANT
	sAmsNetId		: REFERENCE TO T_AmsNetId;
	nAmsPort		: T_AmsPort;
	sInstancePath	: REFERENCE TO STRING;
	sSymbol			: REFERENCE TO STRING;
END_VAR
VAR
	sRpcSymbol : T_MaxString;
END_VAR
IF sAmsNetId = '' THEN
	ConfigDoneCallback := E_HRESULTAdsErr.INVALIDPARM;
	RETURN;
END_IF

IF nAmsPort = 0 THEN
	ConfigDoneCallback := E_HRESULTAdsErr.INVALIDPARM;
	RETURN;
END_IF

IF sInstancePath = '' THEN
	ConfigDoneCallback := E_HRESULTAdsErr.INVALIDPARM;
	RETURN;
END_IF

IF sSymbol = '' THEN
	ConfigDoneCallback := E_HRESULTAdsErr.INVALIDPARM;
	RETURN;
END_IF

IF sAmsNetId <> SUPER^.sAmsNetId THEN
	SUPER^.ReleaseHandle();
	SUPER^.sAmsNetId := sAmsNetId;	
END_IF

IF nAmsPort <> SUPER^.nAmsPort THEN
	SUPER^.ReleaseHandle();
	SUPER^.nAmsPort := nAmsPort;	
END_IF

sRpcSymbol := F_RpcSymbol(sInstancePath:= sInstancePath, sSymbolName:= sSymbol);
IF sRpcSymbol <> SUPER^.sRpcSymbolField THEN
	SUPER^.ReleaseHandle();
	SUPER^.sRpcSymbol := sRpcSymbol;
END_IF;

ConfigDoneCallback := S_OK;
END_METHOD

METHOD Configure : I_RpcDynamicConfigAmsNetId
fbConfig.SetCallback(pFbRpcBase:= THIS);
Configure := fbConfig;
END_METHOD

METHOD FB_exit : BOOL
VAR_INPUT
	bInCopyCode : BOOL; // if TRUE, the exit method is called for exiting an instance that is copied afterwards (online change).
END_VAR
IF SUPER^.nSymbolHandle > cNoSymbolNameHandle THEN
	SUPER^.ReleaseHandle();
END_IF
END_METHOD

END_FUNCTION_BLOCK

// ---- POUs/internal/FB_RpcConfig.TcPOU
{attribute 'no_explicit_call' := 'do not call this POU directly'}
{attribute 'conditionalshow_all_locals'}
FUNCTION_BLOCK INTERNAL FINAL FB_RpcConfig IMPLEMENTS I_RpcDynamicConfigAmsNetId, I_RpcDynamicConfigAmsPort, I_RpcDynamicConfigSymbolPath, I_RpcDynamicConfigBuild
VAR_INPUT
END_VAR
VAR_OUTPUT
END_VAR
VAR	
	sAmsNetIdLocalField		: T_AmsNetId;
	nAmsPortLocalField		: T_AmsPort;
	sInstancePathLocalField	: STRING;
	sSymbolLocalField		: STRING;
	pFbRpcBase				: POINTER TO FB_RpcBase;
END_VAR

METHOD Build : HRESULT
IF pFbRpcBase = NULL THEN
	Build := E_HRESULTAdsErr.INVALIDINTERFACE;
	RETURN;
END_IF
Build := pFbRpcBase^.ConfigDoneCallBack(sAmsNetId:= sAmsNetIdLocalField, nAmsPort:= nAmsPortLocalField, sInstancePath:= sInstancePathLocalField, sSymbol:= sSymbolLocalField);
END_METHOD

METHOD INTERNAL SetCallback
VAR_INPUT
	pFbRpcBase : POINTER TO FB_RpcBase;
END_VAR
THIS^.pFbRpcBase := pFbRpcBase;
END_METHOD

METHOD WithAmsNetId : I_RpcDynamicConfigAmsPort
VAR_INPUT
	sAmsNetId	: Tc2_System.T_AmsNetID;
END_VAR
THIS^.sAmsNetIdLocalField := sAmsNetId;

WithAmsNetId := THIS^;
END_METHOD

METHOD WithAmsPort : I_RpcDynamicConfigSymbolPath
VAR_INPUT
	nAmsPort	: Tc2_System.T_AmsPort;
END_VAR
THIS^.nAmsPortLocalField := nAmsPort;

WithAmsPort := THIS^;
END_METHOD

METHOD WithSymbolPath : I_RpcDynamicConfigBuild
VAR_INPUT
	sInstancePath	: STRING;
	sSymbol	: STRING;
END_VAR
THIS^.sInstancePathLocalField := sInstancePath;
THIS^.sSymbolLocalField := sSymbol;

WithSymbolPath := THIS^;
END_METHOD

END_FUNCTION_BLOCK

// ---- TESTs/FB_F_ToAnyType_Tests.TcPOU
{attribute 'reflection'}
FUNCTION_BLOCK INTERNAL FINAL FB_F_ToAnyType_Tests EXTENDS TcUnit.FB_TestSuite
VAR_INPUT
END_VAR
VAR_OUTPUT
END_VAR
VAR
	{attribute 'instance-path'} 
    {attribute 'noinit'} 
	sTestName			: T_MaxString;
	
	stDummy				: ST_AmsAddr;
	stActual			: ST_AnyType;
END_VAR

TEST(sTestName);

TEST('Should convert __SYSTEM.AnyTpe to ST_AnyType successfully');

// Act
stActual := F_ToAnyType(stDummy);

// Assert
AssertEquals_ULINT(Expected:= ADR(stDummy),
					Actual:= stActual.pValue,
					Message:= 'Pointervalue did not match');
AssertEquals_DINT(Expected:= SIZEOF(stDummy),
					Actual:= stActual.nSize,
					Message:= 'Size did not match');
AssertEquals_DWORD(Expected:= __SYSTEM.TYPE_CLASS.TYPE_USERDEF,
					Actual:= stActual.TypeClass,
					Message:= 'TypeClass did not match');
TEST_FINISHED();

TEST_FINISHED_NAMED(sTestName);

END_FUNCTION_BLOCK
